// TIA Portal V18 export
// export: Created 2025-12-01T12:38:48.2077738Z, ExportSetting None, DisplayName Totally Integrated Automation Portal, DisplayVersion V18 Update 5, DisplayName TIA Portal Openness, DisplayVersion V18 Update 5, DisplayName TIA Portal Teamcenter Gateway, DisplayVersion V18, DisplayName TIA Portal Version Control Interface, DisplayVersion V18, DisplayName STEP 7 Professional, DisplayVersion V18 Update 5, DisplayName STEP 7 Safety, DisplayVersion V18, DisplayName WinCC Professional, DisplayVersion V18 Update 5
FUNCTION "Pilz" : Void   // FC2700, LAD
{ S7_Optimized_Access := 'TRUE' }
// stored: AutoNumber false, SetENOAutomatically false
   VAR_TEMP
      Ret_Val_1 : Int;
      Ret_Val_2 : Int;
      Ret_Val_3 : Int;
      Ret_Val_4 : Int;
   END_VAR
   VAR_TEMP   // added for the SCL form of the ladder/FBD networks
      _w1 : Bool;
   END_VAR
BEGIN

REGION Network 1: 功能块调用 / Pilz
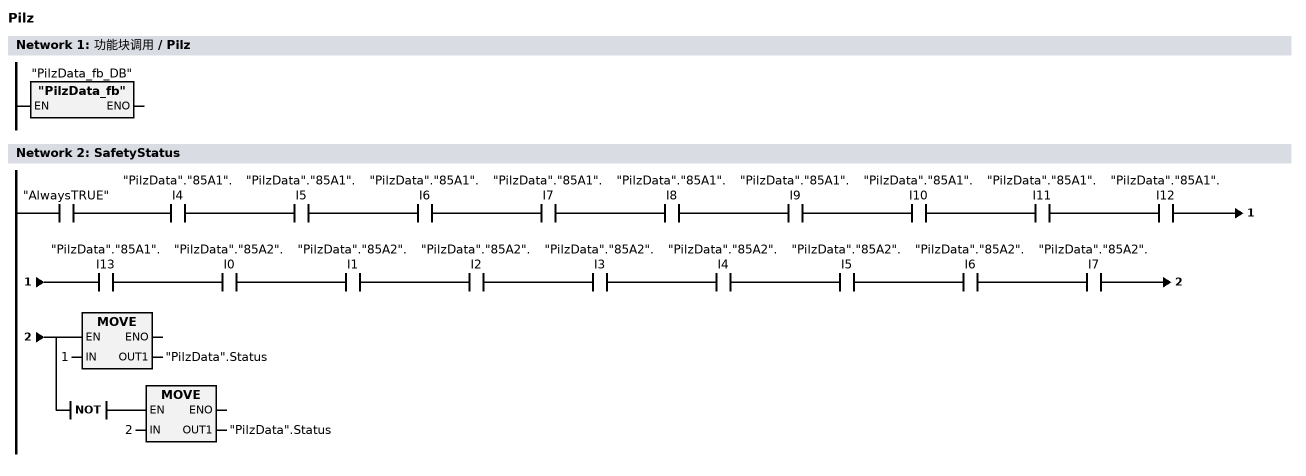
   RUNG wire#powerrail
      "PilzData_fb_DB"()
   END_RUNG
   // the same network as SCL:
   "PilzData_fb_DB"();   // "PilzData_fb"
END_REGION

REGION Network 2: SafetyStatus
   RUNG wire#powerrail
      Contact( "AlwaysTRUE" )
      Contact( "PilzData"."85A1".I4 )
      Contact( "PilzData"."85A1".I5 )
      Contact( "PilzData"."85A1".I6 )
      Contact( "PilzData"."85A1".I7 )
      Contact( "PilzData"."85A1".I8 )
      Contact( "PilzData"."85A1".I9 )
      Contact( "PilzData"."85A1".I10 )
      Contact( "PilzData"."85A1".I11 )
      Contact( "PilzData"."85A1".I12 )
      Contact( "PilzData"."85A1".I13 )
      Contact( "PilzData"."85A2".I0 )
      Contact( "PilzData"."85A2".I1 )
      Contact( "PilzData"."85A2".I2 )
      Contact( "PilzData"."85A2".I3 )
      Contact( "PilzData"."85A2".I4 )
      Contact( "PilzData"."85A2".I5 )
      Contact( "PilzData"."85A2".I6 )
      Contact( "PilzData"."85A2".I7 )
      wire#w1
      Move(in := 1, out1 => "PilzData".Status)
   END_RUNG
   RUNG wire#w1
      Not()
      Move(in := 2, out1 => "PilzData".Status)
   END_RUNG
   // the same network as SCL:
   #_w1 := "AlwaysTRUE" AND "PilzData"."85A1".I4 AND "PilzData"."85A1".I5 AND "PilzData"."85A1".I6 AND "PilzData"."85A1".I7 AND "PilzData"."85A1".I8 AND "PilzData"."85A1".I9 AND "PilzData"."85A1".I10 AND "PilzData"."85A1".I11 AND "PilzData"."85A1".I12 AND "PilzData"."85A1".I13 AND "PilzData"."85A2".I0 AND "PilzData"."85A2".I1 AND "PilzData"."85A2".I2 AND "PilzData"."85A2".I3 AND "PilzData"."85A2".I4 AND "PilzData"."85A2".I5 AND "PilzData"."85A2".I6 AND "PilzData"."85A2".I7;
   IF #_w1 THEN "PilzData".Status := 1; END_IF;
   IF NOT #_w1 THEN "PilzData".Status := 2; END_IF;
END_REGION
END_FUNCTION
